{attribute 'qualified_only'}
VAR_GLOBAL
	Eixo1 : AXIS_REF;
	Eixo2 : AXIS_REF;
END_VAR

(* stored: Version 1.1.0.1
   GVL GVL_Eixos: Id {0a4714c9-f21c-40ab-b947-17dae50dc60a} *)
